(* CODESYS project Dual Magazijn Structured Text 2V0 - Demo 3V5SP13.project
   Company: Avans
   Description: Simulatie voor opstelling Sorteer Station.
   Title: Simulatie Sorteer Station
   Author: Rene Potters/Gerard Harkema
   Version: 0.1.0

Project tree, tasks and I/O mapping:
  Device_1 : CODESYS Control Win V3, 3S - Smart Software Solutions GmbH, version 3.5.13.20
    application MagazijnTestSimulatie
      libraries: Standard, * (System); Util, * (System); VisuDialogs, 3.5.16.40 (System)
      task MainTask (cyclic, interval t#20ms, priority 1) calls MagazijnTest
      task Simulatie (cyclic, interval t#20ms, priority 1) calls MagazijnSim1, MagazijnSim2
  Simulatie/
    program MagazijnSim1 [ST]
    global variables SIM1
    data type MagazijnDUT
    program MagazijnSim2 [ST]
    global variables SIM2
  text list GlobalTextList
  Programma Structured Text/
    function block MagazijnClass [ST]: initialize, cycle, start, isMagazijnLeeg, isError, reset, isKlaar, noodstop
    TestProgramms/
      program MagazijnTest [ST]
    States/
      data type magazijnStates
  global variables GVL1
  Visualisaties/
    visualisation BekerMagazijnHMI
  global variables GVL2
*)

// Simulatie/MagazijnDUT
{attribute 'qualified_only'}
{attribute 'strict'}
TYPE MagazijnDUT :
(
	INGETROKKEN, INTREKKEN, UITGESTOTEN, UITSTOTEN, LEEG
);
END_TYPE

// Programma Structured Text/States/magazijnStates
// Datum : 17 december 2020, Auteur: Gerard Harkema
{attribute 'qualified_only'}
{attribute 'strict'}
TYPE magazijnStates :
(
	idle := 0,
	in,
	travel_out,
	out,
	travel_in,
	error
);
END_TYPE

// Simulatie/SIM1
{attribute 'qualified_only'}
VAR_GLOBAL
	// Rotatie van de overzetter
	Vx_OvzRotate: INT := 0;
	// Visualisatie invisible blok
	Vx_OvzBlokLinks: BOOL := FALSE;
	// Visualisatie invisible blok
	Vx_OvzBlokOverzetter: BOOL := FALSE;
	// Visualisatie invisible blok
	Vx_OvzBlokRechts: BOOL := FALSE;
	// Visualisatie invisible blok
	Vx_OvzBlokGevallen: BOOL := FALSE;	
	// Magazijn opnieuw vullen (simulatie)
	Ix_MagazijnVullen 	: BOOL;
	// Goten legen (symulatie)
	Ix_GotenLegen	  	: BOOL;
	
	
	
	
	
	
	
	
	
	
	
	
	
	
	
	
	
	
	
	
	
	
	
	
	
	
	
	
	
	
	
	
	
	
	
	
	
	
	
	
	
	
	
	
	
	
	
	
	// Simulatie visualisatie 
	Vw_Rotate45: INT := 45;
	// Visualisatie X positie van de uitstoter
	Vw_MagUitstoterBekerX: INT := 30;
	// Visualisatie invisible blok uitgestoten
	Vx_MagBlokUit: BOOL := TRUE;
	// Visualisatie invisible blok 1
	Vx_MagBlok1: BOOL := TRUE;
	// Visualisatie invisible blok 2
	Vx_MagBlok2: BOOL := TRUE;
	// Visualisatie invisible blok 3
	Vx_MagBlok3: BOOL := TRUE;
	// Visualisatie invisible blok 4
	Vx_MagBlok4: BOOL := TRUE;
	// Visualisatie invisible blokken
	Vx_MagBlok: ARRAY[1..8] OF BOOL;
	// Aantal blokken in het magazijn
	Vw_MagBlokAantal: INT := 4;
	// Simulatie onthoudt dat een blok maar 1x wordt uitgestoten
	Vw_MagBlok1X: INT := 0;
	// Ligt er een blok op band
	Vw_SorBlokBand: BOOL := FALSE;
	// Rotatie van de stopper
	Vw_SorStopperRotate: INT := 0;
	// Rotatie van de stopper goot 1
	Vw_SorGoot1Rotate: INT := 0;
	// Rotatie van de stopper goot 2
	Vw_SorGoot2Rotate: INT := 0;
	// Kleur van de blok op betreffende positie
	Vw_SorKleurBand: DWORD := 0;
	// Bewegen van de blok over de band
	Vi_SorBlokBandX: INT := 0;
	// Bewegen van de blok over de band
	Vi_SorBlokBandY: INT := 0;
	// Simulatie error. Inverse logica.
	Vx_MagLuchtDrukError: BOOL := TRUE;
	// Simulatie error. Inverse logica.
	Vx_MagIsInError: BOOL := TRUE;
	// Simulatie error. Inverse logica.
	Vx_MagIsUitError: BOOL := TRUE;
	// Simulatie error. Inverse logica.
	Vx_OvzLuchtDrukError: BOOL := TRUE;
	// Simulatie error. Inverse logica.
	Vx_OvzIsLinksError: BOOL := TRUE;
	// Simulatie error. Inverse logica.
	Vx_OvzIsRechtsError: BOOL := TRUE;
	// Simulatie error. Inverse logica.
	Vx_OvzVacuumError: BOOL := TRUE;
	// Simulatie error. Inverse logica.
	Vx_SorMotorAfvoerError: BOOL := TRUE;
	// Simulatie error. Inverse logica.
	Vx_SorGoot1InError: BOOL := TRUE;
	// Simulatie error. Inverse logica.
	Vx_SorGoot1UitError: BOOL := TRUE;
	// Simulatie error. Inverse logica.
	Vx_SorInGootError: BOOL := TRUE;
	// Ligt er een blok op de betreffende positie
	Vx_SorBlokGoot: ARRAY [1..3,1..6] OF BOOL;
	// Kleur van de blok op betreffende positie
	Vw_SorKleurGoot: ARRAY [1..3,1..6] OF DWORD;
END_VAR

// GVL1
VAR_GLOBAL
	// Indrukken resetknop 
	Ix_Resetknop: BOOL;
	// Keuzeknop staat op hand
	Ix_Hand: BOOL;
	// Keuzeknop staat op auto
	Ix_Auto: BOOL;
	// Indrukken noodstop
	Ix_Noodstop: BOOL;
	// Bekers magazijn zijn op
	Ix_MagazijnLeeg: BOOL;
	// Beker is uit dekselmagazijn gestoten
	Ix_UitstoterBekerIn: BOOL;
	// Uitstoter Beker haalt nieuwe beker op
	Ix_UitstoterBekerUit: BOOL;
	// Indrukken startknop
	Ix_Stopknop: BOOL := TRUE;
	// Indrukken stopknop
	Ix_Startknop: BOOL;	
	//Perslucht is aanwezig
	Ix_PersluchtAanwezig :BOOL;
	//Werkstuk door overzetter opgepakt
	Ix_VacuumAanwezig :BOOL;
	//Overzetter haalt beker op(linker pos.)
	Ix_OverzetterIsLinks :BOOL;
	//Overzetter plaatst beker op sorteerpositie
	Ix_OverzetterIsRechts :BOOL;
	//Beker aanwezig op detectiepositie
	Ix_BekerAanwezig :BOOL;
	//Beker is van aluminium
	Ix_BekerMetaal :BOOL;
	//Beker reflecteert en is dus niet zwart
	Ix_BekerReflecteerd :BOOL;
	//Product is naar een van de goten gegaan
	Ix_BekerInGoot :BOOL;
	//Pusher uitvoergoot 1 is in
	Ix_UitvoerGoot1IsIn :BOOL;
	//Pusher uitvoergoot 2 is in
	Ix_UitvoerGoot2IsIn :BOOL;
	//Beker afvoeren is bezig
	Ix_StationAfvoerVrij :BOOL;
	//Pusher uitvoergoot 1 is uit
	Ix_UitvoerGoot1IsUit :BOOL;
	//Pusher uitvoergoot 2 is uit
	Ix_UitvoerGoot2IsUit :BOOL;
	// Beker uit magazijn stoten
	Qx_BekerUitstoten: BOOL;	
	//Beker oppakken
	Qx_VacuumAan :BOOL;
	//Beker loslaten
	Qx_BekerLossen :BOOL;
	//Overzetter naar bekermagazijn
	Qx_OverzetterLinks :BOOL;
	//Overzetter naar sorteerpositie
	Qx_OverzetterRechts :BOOL;
	//Transportband aan
	Qx_MotorAfvoerAan :BOOL;
	//Pusher goot 1 uit
	Qx_UitvoerGoot1Uit :BOOL;
	//Pusher goot 2 uit
	Qx_UitvoerGoot2Uit :BOOL;
	//Beker stoppen op band voor detectie
	Qx_StopperUit :BOOL;
	//Uitsorteren is bezet
	Qx_StationBezet :BOOL;
	// Visualisatie invisible Gele vlak
	Qx_GeleLamp: BOOL;
	// Visualisatie invisible groene vlak
	Qx_GroeneLamp: BOOL;
	// Visualisatie invisible rode vlak
	Qx_RodeLamp: BOOL;
END_VAR

// Simulatie/SIM2
{attribute 'qualified_only'}
VAR_GLOBAL
	// Rotatie van de overzetter
	Vx_OvzRotate: INT := 0;
	// Visualisatie invisible blok
	Vx_OvzBlokLinks: BOOL := FALSE;
	// Visualisatie invisible blok
	Vx_OvzBlokOverzetter: BOOL := FALSE;
	// Visualisatie invisible blok
	Vx_OvzBlokRechts: BOOL := FALSE;
	// Visualisatie invisible blok
	Vx_OvzBlokGevallen: BOOL := FALSE;	
	// Magazijn opnieuw vullen (simulatie)
	Ix_MagazijnVullen 	: BOOL;
	// Goten legen (symulatie)
	Ix_GotenLegen	  	: BOOL;
	
	
	
	
	
	
	
	
	
	
	
	
	
	
	
	
	
	
	
	
	
	
	
	
	
	
	
	
	
	
	
	
	
	
	
	
	
	
	
	
	
	
	
	
	
	
	
	
	// Simulatie visualisatie 
	Vw_Rotate45: INT := 45;
	// Visualisatie X positie van de uitstoter
	Vw_MagUitstoterBekerX: INT := 30;
	// Visualisatie invisible blok uitgestoten
	Vx_MagBlokUit: BOOL := TRUE;
	// Visualisatie invisible blok 1
	Vx_MagBlok1: BOOL := TRUE;
	// Visualisatie invisible blok 2
	Vx_MagBlok2: BOOL := TRUE;
	// Visualisatie invisible blok 3
	Vx_MagBlok3: BOOL := TRUE;
	// Visualisatie invisible blok 4
	Vx_MagBlok4: BOOL := TRUE;
	// Visualisatie invisible blokken
	Vx_MagBlok: ARRAY[1..8] OF BOOL;
	// Aantal blokken in het magazijn
	Vw_MagBlokAantal: INT := 4;
	// Simulatie onthoudt dat een blok maar 1x wordt uitgestoten
	Vw_MagBlok1X: INT := 0;
	// Ligt er een blok op band
	Vw_SorBlokBand: BOOL := FALSE;
	// Rotatie van de stopper
	Vw_SorStopperRotate: INT := 0;
	// Rotatie van de stopper goot 1
	Vw_SorGoot1Rotate: INT := 0;
	// Rotatie van de stopper goot 2
	Vw_SorGoot2Rotate: INT := 0;
	// Kleur van de blok op betreffende positie
	Vw_SorKleurBand: DWORD := 0;
	// Bewegen van de blok over de band
	Vi_SorBlokBandX: INT := 0;
	// Bewegen van de blok over de band
	Vi_SorBlokBandY: INT := 0;
	// Simulatie error. Inverse logica.
	Vx_MagLuchtDrukError: BOOL := TRUE;
	// Simulatie error. Inverse logica.
	Vx_MagIsInError: BOOL := TRUE;
	// Simulatie error. Inverse logica.
	Vx_MagIsUitError: BOOL := TRUE;
	// Simulatie error. Inverse logica.
	Vx_OvzLuchtDrukError: BOOL := TRUE;
	// Simulatie error. Inverse logica.
	Vx_OvzIsLinksError: BOOL := TRUE;
	// Simulatie error. Inverse logica.
	Vx_OvzIsRechtsError: BOOL := TRUE;
	// Simulatie error. Inverse logica.
	Vx_OvzVacuumError: BOOL := TRUE;
	// Simulatie error. Inverse logica.
	Vx_SorMotorAfvoerError: BOOL := TRUE;
	// Simulatie error. Inverse logica.
	Vx_SorGoot1InError: BOOL := TRUE;
	// Simulatie error. Inverse logica.
	Vx_SorGoot1UitError: BOOL := TRUE;
	// Simulatie error. Inverse logica.
	Vx_SorInGootError: BOOL := TRUE;
	// Ligt er een blok op de betreffende positie
	Vx_SorBlokGoot: ARRAY [1..3,1..6] OF BOOL;
	// Kleur van de blok op betreffende positie
	Vw_SorKleurGoot: ARRAY [1..3,1..6] OF DWORD;
END_VAR

// GVL2
VAR_GLOBAL
	// Indrukken resetknop 
	Ix_Resetknop: BOOL;
	// Keuzeknop staat op hand
	Ix_Hand: BOOL;
	// Keuzeknop staat op auto
	Ix_Auto: BOOL;
	// Indrukken noodstop
	Ix_Noodstop: BOOL;
	// Bekers magazijn zijn op
	Ix_MagazijnLeeg: BOOL;
	// Beker is uit dekselmagazijn gestoten
	Ix_UitstoterBekerIn: BOOL;
	// Uitstoter Beker haalt nieuwe beker op
	Ix_UitstoterBekerUit: BOOL;
	// Indrukken startknop
	Ix_Stopknop: BOOL := TRUE;
	// Indrukken stopknop
	Ix_Startknop: BOOL;	
	//Perslucht is aanwezig
	Ix_PersluchtAanwezig :BOOL;
	//Werkstuk door overzetter opgepakt
	Ix_VacuumAanwezig :BOOL;
	//Overzetter haalt beker op(linker pos.)
	Ix_OverzetterIsLinks :BOOL;
	//Overzetter plaatst beker op sorteerpositie
	Ix_OverzetterIsRechts :BOOL;
	//Beker aanwezig op detectiepositie
	Ix_BekerAanwezig :BOOL;
	//Beker is van aluminium
	Ix_BekerMetaal :BOOL;
	//Beker reflecteert en is dus niet zwart
	Ix_BekerReflecteerd :BOOL;
	//Product is naar een van de goten gegaan
	Ix_BekerInGoot :BOOL;
	//Pusher uitvoergoot 1 is in
	Ix_UitvoerGoot1IsIn :BOOL;
	//Pusher uitvoergoot 2 is in
	Ix_UitvoerGoot2IsIn :BOOL;
	//Beker afvoeren is bezig
	Ix_StationAfvoerVrij :BOOL;
	//Pusher uitvoergoot 1 is uit
	Ix_UitvoerGoot1IsUit :BOOL;
	//Pusher uitvoergoot 2 is uit
	Ix_UitvoerGoot2IsUit :BOOL;
	// Beker uit magazijn stoten
	Qx_BekerUitstoten: BOOL;	
	//Beker oppakken
	Qx_VacuumAan :BOOL;
	//Beker loslaten
	Qx_BekerLossen :BOOL;
	//Overzetter naar bekermagazijn
	Qx_OverzetterLinks :BOOL;
	//Overzetter naar sorteerpositie
	Qx_OverzetterRechts :BOOL;
	//Transportband aan
	Qx_MotorAfvoerAan :BOOL;
	//Pusher goot 1 uit
	Qx_UitvoerGoot1Uit :BOOL;
	//Pusher goot 2 uit
	Qx_UitvoerGoot2Uit :BOOL;
	//Beker stoppen op band voor detectie
	Qx_StopperUit :BOOL;
	//Uitsorteren is bezet
	Qx_StationBezet :BOOL;
	// Visualisatie invisible Gele vlak
	Qx_GeleLamp: BOOL;
	// Visualisatie invisible groene vlak
	Qx_GroeneLamp: BOOL;
	// Visualisatie invisible rode vlak
	Qx_RodeLamp: BOOL;
END_VAR

// Programma Structured Text/TestProgramms/MagazijnTest
// Datum : 17 december 2020, Auteur: Gerard Harkema
PROGRAM MagazijnTest
VAR
	xInitialaized				: BOOL := FALSE;
	
	// Bekers magazijn zijn op
	Ix_MagazijnLeegRef1			: REFERENCE TO BOOL;
	// Beker is uit dekselmagazijn gestoten
	Ix_UitstoterBekerInRef1		: REFERENCE TO BOOL;
	// Uitstoter Beker haalt nieuwe beker op
	Ix_UitstoterBekerUitRef1	: REFERENCE TO BOOL;
	// Beker uit magazijn stoten
	Qx_BekerUitstotenRef1		: REFERENCE TO BOOL;
	
	// Bekers magazijn zijn op
	Ix_MagazijnLeegRef2			: REFERENCE TO BOOL;
	// Beker is uit dekselmagazijn gestoten
	Ix_UitstoterBekerInRef2		: REFERENCE TO BOOL;
	// Uitstoter Beker haalt nieuwe beker op
	Ix_UitstoterBekerUitRef2	: REFERENCE TO BOOL;
	// Beker uit magazijn stoten
	Qx_BekerUitstotenRef2		: REFERENCE TO BOOL;

	magazijn1: MagazijnClass;
	magazijn2: MagazijnClass;
	
END_VAR

IF NOT xInitialaized THEN

	// Forse Persluct aanwezig
	GVL1.Ix_PersluchtAanwezig := TRUE;
	
	Ix_MagazijnLeegRef1 		REF= GVL1.Ix_MagazijnLeeg;
	Ix_UitstoterBekerInRef1 	REF= GVL1.Ix_UitstoterBekerIn;
	Ix_UitstoterBekerUitRef1 	REF= GVL1.Ix_UitstoterBekerUit;
	Qx_BekerUitstotenRef1 		REF= GVL1.Qx_BekerUitstoten;

	magazijn1.initialize(Ix_MagazijnLeegRef1,
					    Ix_UitstoterBekerInRef1,
						Ix_UitstoterBekerUitRef1,
						Qx_BekerUitstotenRef1,
						GVL1.Ix_PersluchtAanwezig);
	
	Ix_MagazijnLeegRef2 		REF= GVL2.Ix_MagazijnLeeg;
	Ix_UitstoterBekerInRef2 	REF= GVL2.Ix_UitstoterBekerIn;
	Ix_UitstoterBekerUitRef2 	REF= GVL2.Ix_UitstoterBekerUit;
	Qx_BekerUitstotenRef2 		REF= GVL2.Qx_BekerUitstoten;

	magazijn2.initialize(Ix_MagazijnLeegRef2,
					    Ix_UitstoterBekerInRef2,
						Ix_UitstoterBekerUitRef2,
						Qx_BekerUitstotenRef2,
						GVL1.Ix_PersluchtAanwezig);
						
						
	xInitialaized	:= TRUE;
END_IF

IF GVL1.Ix_Startknop THEN
	magazijn1.start();
	GVL1.Ix_Startknop := FALSE;
END_IF

IF GVL1.Ix_Resetknop THEN
	magazijn1.reset();
END_IF

IF GVL1.Ix_Noodstop THEN
	magazijn1.noodstop();
END_IF

GVL1.Qx_GroeneLamp := magazijn1.isKlaar();
GVL1.Qx_RodeLamp := magazijn1.isError();
GVL1.Qx_GeleLamp := magazijn1.isMagazijnLeeg();
 
IF GVL2.Ix_Startknop THEN
	magazijn2.start();
	GVL2.Ix_Startknop := FALSE;
END_IF

IF GVL2.Ix_Resetknop THEN
	magazijn2.reset();
END_IF

IF GVL2.Ix_Noodstop THEN
	magazijn2.noodstop();
END_IF

GVL2.Qx_GroeneLamp := magazijn2.isKlaar();
GVL2.Qx_RodeLamp := magazijn2.isError();
GVL2.Qx_GeleLamp := magazijn2.isMagazijnLeeg();

magazijn1.cycle();
magazijn2.cycle();

END_PROGRAM

// Programma Structured Text/MagazijnClass
// Datum : 17 december 2020, Auteur: Gerard Harkema
FUNCTION_BLOCK MagazijnClass
VAR
	// Bekers magazijn zijn op
	Ix_MagazijnLeeg				: REFERENCE TO BOOL;
	// Beker is uit dekselmagazijn gestoten
	Ix_UitstoterBekerIn			: REFERENCE TO BOOL;
	// Uitstoter Beker haalt nieuwe beker op
	Ix_UitstoterBekerUit		: REFERENCE TO BOOL;
	// Beker uit magazijn stoten
	Qx_BekerUitstoten			: REFERENCE TO BOOL;

	//Perslucht is aanwezig
	Ix_PersluchtAanwezig 		: REFERENCE TO BOOL;

	xInitialized				: BOOL := FALSE;
	xKlaar						: BOOL := FALSE;
	eState 						: magazijnStates := magazijnStates.idle;
	
END_VAR

IF NOT xInitialized THEN

	xInitialized				:= TRUE;

END_IF

// Datum : 17 december 2020, Auteur: Gerard Harkema
METHOD initialize
VAR_INPUT
	// Bekers magazijn zijn op
	Ix_MagazijnLeegRef		: REFERENCE TO BOOL;
	// Beker is uit dekselmagazijn gestoten
	Ix_UitstoterBekerInRef	: REFERENCE TO BOOL;
	// Uitstoter Beker haalt nieuwe beker op
	Ix_UitstoterBekerUitRef	: REFERENCE TO BOOL;
	// Beker uit magazijn stoten
	Qx_BekerUitstotenRef	: REFERENCE TO BOOL;
	
	//Perslucht is aanwezig
	Ix_PersluchtAanwezigRef : REFERENCE TO BOOL;

END_VAR
// Bekers magazijn zijn op
Ix_MagazijnLeeg 			REF= Ix_MagazijnLeegRef;
// Beker is uit dekselmagazijn gestoten
Ix_UitstoterBekerIn 		REF= Ix_UitstoterBekerInRef;
// Uitstoter Beker haalt nieuwe beker op
Ix_UitstoterBekerUit 		REF= Ix_UitstoterBekerUitRef;
// Beker uit magazijn stoten
Qx_BekerUitstoten 			REF= Qx_BekerUitstotenRef;
//Perslucht is aanwezig
Ix_PersluchtAanwezig 		REF= Ix_PersluchtAanwezigRef;

eState 						:= magazijnStates.travel_in;
END_METHOD

// Datum : 17 december 2020, Auteur: Gerard Harkema
METHOD cycle
VAR_INPUT
END_VAR

CASE eState OF
	//magazijnStates.idle:
	//magazijnStates.in:
	magazijnStates.travel_out:
		IF Ix_UitstoterBekerUit THEN
			eState 			:= magazijnStates.out;	
			Qx_BekerUitstoten 	:= FALSE;
		END_IF
	magazijnStates.out:
		eState 				:= magazijnStates.travel_in;	
	magazijnStates.travel_in:
		IF Ix_UitstoterBekerIn THEN
			eState 			:= magazijnStates.in;
			xKlaar			:= True;	
		END_IF
	
	//magazijnStates.error:
END_CASE
END_METHOD

// Datum : 17 december 2020, Auteur: Gerard Harkema
METHOD start : BOOL
VAR_INPUT
END_VAR
IF isMagazijnLeeg() THEN
	eState 				:= magazijnStates.error;
	Qx_BekerUitstoten 	:= FALSE;
	start 		:= TRUE; // Failed
	RETURN;
END_IF

IF NOT Ix_PersluchtAanwezig THEN
	eState 				:= magazijnStates.error;
	Qx_BekerUitstoten 	:= FALSE;
	start 		:= TRUE; // Failed
	RETURN;
END_IF

IF NOT (eState = magazijnStates.in) THEN
	eState 				:= magazijnStates.error;
	Qx_BekerUitstoten 	:= FALSE;
	start 		:= TRUE; // Failed
	RETURN;	
END_IF

xKlaar 					:= FALSE;
Qx_BekerUitstoten 		:= TRUE;
eState 					:= magazijnStates.travel_out;

start 			:= FALSE; // oké
END_METHOD

// Datum : 17 december 2020, Auteur: Gerard Harkema
METHOD isMagazijnLeeg : BOOL
VAR_INPUT
END_VAR
isMagazijnLeeg := Ix_MagazijnLeeg;
END_METHOD

// Datum : 17 december 2020, Auteur: Gerard Harkema
METHOD isError : BOOL
VAR_INPUT
END_VAR
isError := (eState = magazijnStates.error);
END_METHOD

// Datum : 17 december 2020, Auteur: Gerard Harkema
METHOD reset : BOOL
VAR_INPUT
END_VAR
eState 		:= magazijnStates.travel_in;
END_METHOD

// Datum : 17 december 2020, Auteur: Gerard Harkema
METHOD isKlaar : BOOL
VAR_INPUT
END_VAR
isKlaar := xKlaar;
END_METHOD

// Datum : 17 december 2020, Auteur: Gerard Harkema
METHOD noodstop
VAR_INPUT
END_VAR
eState 				:= magazijnStates.error;
Qx_BekerUitstoten 	:= FALSE;
END_METHOD

END_FUNCTION_BLOCK

// Simulatie/MagazijnSim1
PROGRAM MagazijnSim1
VAR
	// Timer om uitstoten en intrekken te vertragen
	Fb_Pulse: BLINK;
	// Timer om intrekken te vertragen
	Fb_Trigger: F_TRIG;
	// Eerste keer om visualisatie te updaten
	Mx_FirstTime: BOOL := TRUE;
	// Afhandeling van het magazijn
	Me_MagState: MAGAZIJNDUT := MAGAZIJNDUT.INGETROKKEN;
END_VAR

//
// Common stuff.
//

IF (Mx_FirstTime) THEN
	SIM1.Vw_MagBlokAantal := 8;
	SIM1.Vx_MagBlokUit:= FALSE;
	
	Mx_FirstTime := FALSE;
END_IF

					
//
// Handle all pulse and trigger events.
//
Fb_Pulse(ENABLE:=TRUE,TIMELOW:=T#200MS, TIMEHIGH:=T#200MS);
Fb_Trigger(CLK:=Fb_Pulse.OUT);


//
// Only if no emergency active, start handling the simulation.
//
IF (SIM1.Ix_MagazijnVullen) THEN
	Mx_FirstTime := TRUE;
	SIM1.Ix_MagazijnVullen := FALSE;
	RETURN;
END_IF
	
//
// The pulse determines the speed of the cilinder to move in
// ore move out. The cilinder is only moved if the airpressure 
// is available.
//
IF (Fb_Trigger.Q AND SIM1.Vx_MagLuchtDrukError) THEN
		
			
	CASE Me_MagState OF
		MAGAZIJNDUT.INGETROKKEN:
			IF (SIM1.Vx_MagBlokUit) THEN
				SIM1.Vw_MagBlokAantal := SIM1.Vw_MagBlokAantal - 1;
			END_IF
		
			SIM1.Vw_MagUitstoterBekerX := 1;
			SIM1.Vw_MagBlok1X    	  := SIM1.Vw_MagUitstoterBekerX;
			SIM1.Vx_MagBlokUit         := FALSE;
	
			IF (GVL1.Qx_BekerUitstoten) THEN
				Me_MagState := MAGAZIJNDUT.UITSTOTEN;
			END_IF

		MAGAZIJNDUT.INTREKKEN:
			SIM1.Vw_MagUitstoterBekerX := SIM1.Vw_MagUitstoterBekerX - 30;
			
			IF (SIM1.Vw_MagUitstoterBekerX < 0) THEN 
				SIM1.Vw_MagUitstoterBekerX := 0; 
			END_IF		
			
			IF (SIM1.Vw_MagUitstoterBekerX = 0) THEN
				Me_MagState := MAGAZIJNDUT.INGETROKKEN;				
			END_IF		

			IF (GVL1.Qx_BekerUitstoten) THEN
				Me_MagState := MAGAZIJNDUT.UITSTOTEN;
			END_IF	
	
		MAGAZIJNDUT.UITGESTOTEN:
			SIM1.Vx_MagBlokUit         := SIM1.Vx_MagBlok1;
						
			IF (NOT GVL1.Qx_BekerUitstoten) THEN
				Me_MagState := MAGAZIJNDUT.INTREKKEN;
			END_IF	
		
		MAGAZIJNDUT.UITSTOTEN:
			SIM1.Vw_MagUitstoterBekerX := SIM1.Vw_MagUitstoterBekerX + 30;
			SIM1.Vw_MagBlok1X    	  := SIM1.Vw_MagUitstoterBekerX;			
		
			IF (SIM1.Vw_MagUitstoterBekerX > 70) THEN
				Me_MagState := MAGAZIJNDUT.UITGESTOTEN;				
			END_IF		

			IF (NOT GVL1.Qx_BekerUitstoten) THEN
				Me_MagState := MAGAZIJNDUT.INTREKKEN;
			END_IF	
		
	END_CASE

	GVL1.Ix_UitstoterBekerIn  := (Me_MagState = MAGAZIJNDUT.INGETROKKEN) AND SIM1.Vx_MagIsInError;
	GVL1.Ix_UitstoterBekerUit := (Me_MagState = MAGAZIJNDUT.UITGESTOTEN) AND SIM1.Vx_MagIsUitError;	
	GVL1.Ix_MagazijnLeeg 	 := (SIM1.Vw_MagBlokAantal <= 0) AND (GVL1.Ix_UitstoterBekerIn);	
	
	SIM1.Vx_MagBlok[8] := (SIM1.Vw_MagBlokAantal >= 8);
	SIM1.Vx_MagBlok[7] := (SIM1.Vw_MagBlokAantal >= 7);
	SIM1.Vx_MagBlok[6] := (SIM1.Vw_MagBlokAantal >= 6);
	SIM1.Vx_MagBlok[5] := (SIM1.Vw_MagBlokAantal >= 5);		
	SIM1.Vx_MagBlok[4] := (SIM1.Vw_MagBlokAantal >= 4);
	SIM1.Vx_MagBlok[3] := (SIM1.Vw_MagBlokAantal >= 3);
	SIM1.Vx_MagBlok[2] := (SIM1.Vw_MagBlokAantal >= 2);
	SIM1.Vx_MagBlok[1] := (SIM1.Vw_MagBlokAantal >= 1);	
	
END_IF

END_PROGRAM

// Simulatie/MagazijnSim2
PROGRAM MagazijnSim2
VAR
	// Timer om uitstoten en intrekken te vertragen
	Fb_Pulse: BLINK;
	// Timer om intrekken te vertragen
	Fb_Trigger: F_TRIG;
	// Eerste keer om visualisatie te updaten
	Mx_FirstTime: BOOL := TRUE;
	// Afhandeling van het magazijn
	Me_MagState: MAGAZIJNDUT := MAGAZIJNDUT.INGETROKKEN;
END_VAR

//
// Common stuff.
//

IF (Mx_FirstTime) THEN
	SIM2.Vw_MagBlokAantal := 8;
	SIM2.Vx_MagBlokUit:= FALSE;
	
	Mx_FirstTime := FALSE;
END_IF

					
//
// Handle all pulse and trigger events.
//
Fb_Pulse(ENABLE:=TRUE,TIMELOW:=T#200MS, TIMEHIGH:=T#200MS);
Fb_Trigger(CLK:=Fb_Pulse.OUT);


//
// Only if no emergency active, start handling the simulation.
//
IF (SIM2.Ix_MagazijnVullen) THEN
	Mx_FirstTime := TRUE;
	SIM2.Ix_MagazijnVullen := FALSE;
	RETURN;
END_IF
	
//
// The pulse determines the speed of the cilinder to move in
// ore move out. The cilinder is only moved if the airpressure 
// is available.
//
IF (Fb_Trigger.Q AND SIM2.Vx_MagLuchtDrukError) THEN
		
			
	CASE Me_MagState OF
		MAGAZIJNDUT.INGETROKKEN:
			IF (SIM2.Vx_MagBlokUit) THEN
				SIM2.Vw_MagBlokAantal := SIM2.Vw_MagBlokAantal - 1;
			END_IF
		
			SIM2.Vw_MagUitstoterBekerX := 1;
			SIM2.Vw_MagBlok1X    	  := SIM2.Vw_MagUitstoterBekerX;
			SIM2.Vx_MagBlokUit         := FALSE;
	
			IF (GVL2.Qx_BekerUitstoten) THEN
				Me_MagState := MAGAZIJNDUT.UITSTOTEN;
			END_IF

		MAGAZIJNDUT.INTREKKEN:
			SIM2.Vw_MagUitstoterBekerX := SIM2.Vw_MagUitstoterBekerX - 30;
			
			IF (SIM2.Vw_MagUitstoterBekerX < 0) THEN 
				SIM2.Vw_MagUitstoterBekerX := 0; 
			END_IF		
			
			IF (SIM2.Vw_MagUitstoterBekerX = 0) THEN
				Me_MagState := MAGAZIJNDUT.INGETROKKEN;				
			END_IF		

			IF (GVL2.Qx_BekerUitstoten) THEN
				Me_MagState := MAGAZIJNDUT.UITSTOTEN;
			END_IF	
	
		MAGAZIJNDUT.UITGESTOTEN:
			SIM2.Vx_MagBlokUit         := SIM2.Vx_MagBlok1;
						
			IF (NOT GVL2.Qx_BekerUitstoten) THEN
				Me_MagState := MAGAZIJNDUT.INTREKKEN;
			END_IF	
		
		MAGAZIJNDUT.UITSTOTEN:
			SIM2.Vw_MagUitstoterBekerX := SIM2.Vw_MagUitstoterBekerX + 30;
			SIM2.Vw_MagBlok1X    	  := SIM2.Vw_MagUitstoterBekerX;			
		
			IF (SIM2.Vw_MagUitstoterBekerX > 70) THEN
				Me_MagState := MAGAZIJNDUT.UITGESTOTEN;				
			END_IF		

			IF (NOT GVL2.Qx_BekerUitstoten) THEN
				Me_MagState := MAGAZIJNDUT.INTREKKEN;
			END_IF	
		
	END_CASE

	GVL2.Ix_UitstoterBekerIn  := (Me_MagState = MAGAZIJNDUT.INGETROKKEN) AND SIM2.Vx_MagIsInError;
	GVL2.Ix_UitstoterBekerUit := (Me_MagState = MAGAZIJNDUT.UITGESTOTEN) AND SIM2.Vx_MagIsUitError;	
	GVL2.Ix_MagazijnLeeg 	 := (SIM2.Vw_MagBlokAantal <= 0) AND (GVL2.Ix_UitstoterBekerIn);	
	
	SIM2.Vx_MagBlok[8] := (SIM2.Vw_MagBlokAantal >= 8);
	SIM2.Vx_MagBlok[7] := (SIM2.Vw_MagBlokAantal >= 7);
	SIM2.Vx_MagBlok[6] := (SIM2.Vw_MagBlokAantal >= 6);
	SIM2.Vx_MagBlok[5] := (SIM2.Vw_MagBlokAantal >= 5);		
	SIM2.Vx_MagBlok[4] := (SIM2.Vw_MagBlokAantal >= 4);
	SIM2.Vx_MagBlok[3] := (SIM2.Vw_MagBlokAantal >= 3);
	SIM2.Vx_MagBlok[2] := (SIM2.Vw_MagBlokAantal >= 2);
	SIM2.Vx_MagBlok[1] := (SIM2.Vw_MagBlokAantal >= 1);	
	
END_IF

END_PROGRAM

// Visualisaties/BekerMagazijnHMI
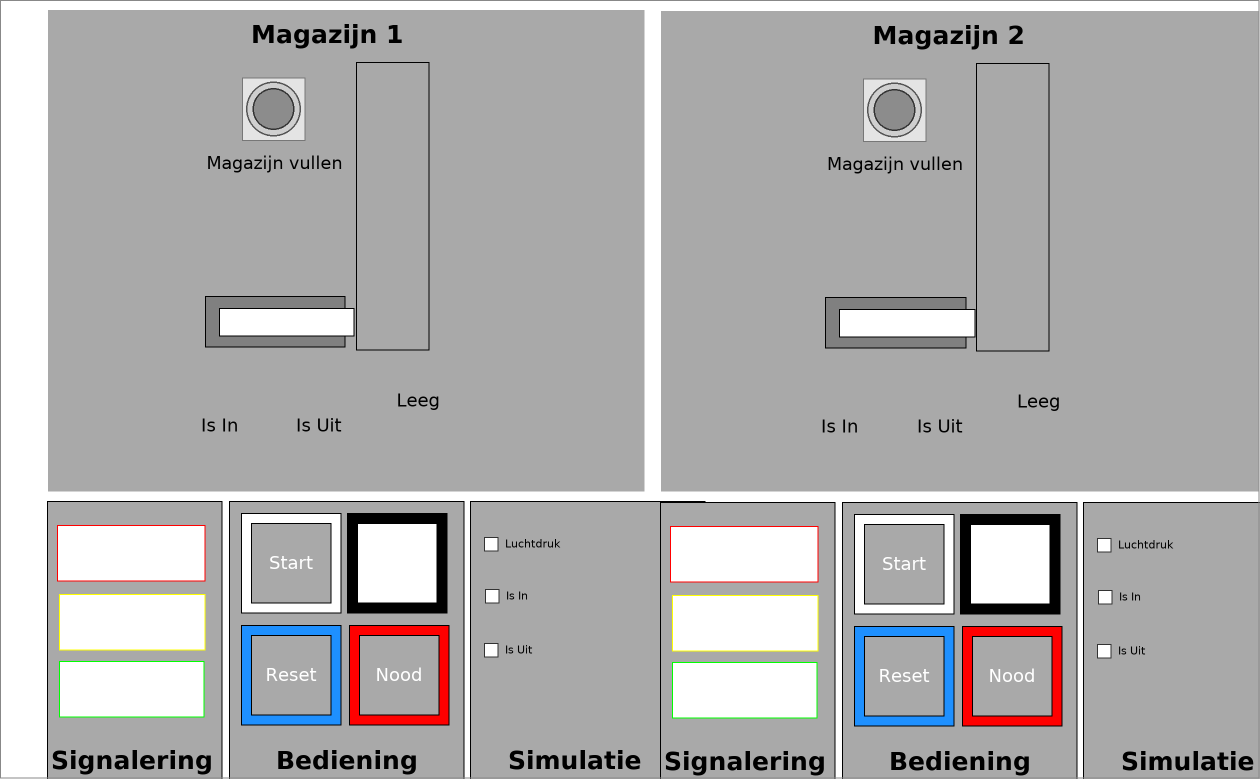
VISUALIZATION BekerMagazijnHMI  // 1260x779
    Group (47,9 1213x770)
        Group (0,0 599x769)
            Group (0,492 599x277)
                Group (0,0 173x277)
                    Rectangle (0,0 175x295)
                    Rectangle (10,24 148x56), colour toggle: GVL1.Qx_RodeLamp
                    Rectangle (12,93 146x56), colour toggle: GVL1.Qx_GeleLamp
                    Rectangle (12,160 145x56), colour toggle: GVL1.Qx_GroeneLamp
                    Label (10,236 150x46), "Signalering"
                Group (182,0 232x277)
                    Rectangle (0,0 235x295)
                    Group (12,12 100x100)
                        RoundedRectangle (0,0 100x100)
                        RoundedRectangle (10,10 80x80), "Start", tooltip "Start knop", colour toggle: GVL1.Ix_Startknop
                            OnMouseDown: execute { gvl1.Ix_Startknop := TRUE; }
                            OnMouseUp: execute { GVL1.Ix_Startknop := FALSE; }
                    Group (118,12 100x100)
                        RoundedRectangle (0,0 100x100)
                        RoundedRectangle (10,10 80x80), "Stop", tooltip "Stop knop", colour toggle: GVL1.Ix_Stopknop
                            OnMouseDown: execute { GVL1.Ix_Stopknop := FALSE; }
                            OnMouseUp: execute { GVL1.Ix_Stopknop := TRUE; }
                    Group (12,124 100x100)
                        RoundedRectangle (0,0 100x100)
                        RoundedRectangle (10,10 80x80), "Reset", tooltip "Reset knop", colour toggle: GVL1.Ix_Resetknop
                            OnMouseUp: execute { GVL1.Ix_Resetknop := FALSE; }
                    Group (120,124 100x100)
                        RoundedRectangle (0,0 100x100), "Nood"
                        RoundedRectangle (10,10 80x80), "Nood", tooltip "Noodstop", colour toggle: GVL1.Ix_Noodstop
                            OnMouseDown: execute { GVL1.Ix_Noodstop := NOT GVL1.Ix_Noodstop; }
                    Label (43,236 150x46), "Bediening"
                Group (423,0 176x277)
                    Group (0,0 235x295)
                        Rectangle (0,0 235x295)
                        Label (30,236 150x46), "Simulatie"
                    Checkbox (12,17 196x52), "Luchtdruk", variable: SIM1.Vx_MagLuchtDrukError
                    Checkbox (13,69 196x52), "Is In", variable: SIM1.Vx_MagIsInError
                    Checkbox (12,123 196x52), "Is Uit", variable: SIM1.Vx_MagIsUitError
            Group (0,0 598x483)
                Rectangle (0,0 598x483)
                Polygon (331,379) (358,379) (385,379) (412,379) (371,454), "Leeg", colour toggle: GVL1.Ix_MagazijnLeeg
                Polygon (173,379) (173,379) (209,417) (173,454) (137,417), "Is In", colour toggle: GVL1.Ix_UitstoterBekerIn
                Polygon (272,379) (272,379) (308,417) (272,454) (236,417), "Is Uit", colour toggle: GVL1.Ix_UitstoterBekerUit
                Rectangle (158,287 140x51)
                Rectangle (309,53 73x288)
                Rectangle (392,300 55x27), colour toggle: SIM1.Vx_MagBlokUit
                Rectangle (313,267 55x27), colour toggle: SIM1.Vx_MagBlok[2]
                Rectangle (313,233 55x27), colour toggle: SIM1.Vx_MagBlok[3]
                Rectangle (313,199 55x27), colour toggle: SIM1.Vx_MagBlok[4]
                Rectangle (313,300 55x27), colour toggle: SIM1.Vx_MagBlok[1]
                    p3560616238: SIM1.Vw_MagBlok1X
                Rectangle (172,299 135x28)
                    p3560616238: SIM1.Vw_MagUitstoterBekerX
                Label (213,11 135x28), "Magazijn 1"
                Rectangle (313,132 55x27), colour toggle: SIM1.Vx_MagBlok[6]
                Rectangle (313,98 55x27), colour toggle: SIM1.Vx_MagBlok[7]
                Rectangle (313,64 55x27), colour toggle: SIM1.Vx_MagBlok[8]
                Rectangle (313,165 55x27), colour toggle: SIM1.Vx_MagBlok[5]
                PushSwitch (195,67 63x66), tooltip "Magazijn vullen", variable: SIM1.Ix_MagazijnVullen, behaviour: TOGGLE, style: Switch-PushSwitch-Gray
                Polygon (158,142) (185,142) (212,142) (297,156) (207,169), "Magazijn vullen", colour toggle: Ix_MagazijnLeeg
        Group (613,1 600x769)
            Group (0,492 600x277)
                Group (0,0 173x277)
                    Rectangle (0,0 175x295)
                    Rectangle (10,24 148x56), colour toggle: GVL2.Qx_RodeLamp
                    Rectangle (12,93 146x56), colour toggle: GVL2.Qx_GeleLamp
                    Rectangle (12,160 145x56), colour toggle: GVL2.Qx_GroeneLamp
                    Label (10,236 150x46), "Signalering"
                Group (182,0 232x277)
                    Rectangle (0,0 235x295)
                    Group (12,12 100x100)
                        RoundedRectangle (0,0 100x100)
                        RoundedRectangle (10,10 80x80), "Start", tooltip "Start knop", colour toggle: GVL2.Ix_Startknop
                            OnMouseDown: execute { GVL2.Ix_Startknop := TRUE; }
                            OnMouseUp: execute { GVL2.Ix_Startknop := FALSE; }
                    Group (118,12 100x100)
                        RoundedRectangle (0,0 100x100)
                        RoundedRectangle (10,10 80x80), "Stop", tooltip "Stop knop", colour toggle: GVL2.Ix_Stopknop
                            OnMouseDown: execute { GVL2.Ix_Stopknop := FALSE; }
                            OnMouseUp: execute { GVL2.Ix_Stopknop := TRUE; }
                    Group (12,124 100x100)
                        RoundedRectangle (0,0 100x100)
                        RoundedRectangle (10,10 80x80), "Reset", tooltip "Reset knop", colour toggle: GVL2.Ix_Resetknop
                            OnMouseDown: execute { GVL2.Ix_Resetknop := TRUE; }
                            OnMouseUp: execute { GVL2.Ix_Resetknop := FALSE; }
                    Group (120,124 100x100)
                        RoundedRectangle (0,0 100x100), "Nood"
                        RoundedRectangle (10,10 80x80), "Nood", tooltip "Noodstop", colour toggle: GVL2.Ix_Noodstop
                            OnMouseDown: execute { Ix_Noodstop := NOT Ix_Noodstop; }
                    Label (43,236 150x46), "Bediening"
                Group (423,0 177x277)
                    Rectangle (0,0 235x295)
                    Label (30,236 150x46), "Simulatie"
                    Checkbox (12,17 196x52), "Luchtdruk", variable: SIM2.Vx_MagLuchtDrukError
                    Checkbox (13,69 196x52), "Is In", variable: SIM2.Vx_MagIsInError
                    Checkbox (12,123 196x52), "Is Uit", variable: SIM2.Vx_MagIsUitError
            Group (0,0 600x482)
                Rectangle (0,0 600x482)
                Polygon (338,379) (366,379) (393,379) (420,379) (379,454), "Leeg", colour toggle: GVL2.Ix_MagazijnLeeg
                Polygon (180,379) (180,379) (216,417) (180,454) (144,417), "Is In", colour toggle: GVL2.Ix_UitstoterBekerIn
                Polygon (280,379) (280,379) (316,417) (280,454) (244,417), "Is Uit", colour toggle: GVL2.Ix_UitstoterBekerUit
                Rectangle (165,287 141x51)
                Rectangle (316,53 73x288)
                Rectangle (400,300 55x27), colour toggle: SIM2.Vx_MagBlokUit
                Rectangle (321,267 55x27), colour toggle: SIM2.Vx_MagBlok[2]
                Rectangle (321,233 55x27), colour toggle: SIM2.Vx_MagBlok[3]
                Rectangle (321,199 55x27), colour toggle: SIM2.Vx_MagBlok[4]
                Rectangle (321,300 55x27), colour toggle: SIM2.Vx_MagBlok[1]
                    p3560616238: SIM2.Vw_MagBlok1X
                Rectangle (179,299 136x28)
                    p3560616238: SIM2.Vw_MagUitstoterBekerX
                Label (214,11 150x28), "Magazijn 2"
                Rectangle (321,132 55x27), colour toggle: SIM2.Vx_MagBlok[6]
                Rectangle (321,98 55x27), colour toggle: SIM2.Vx_MagBlok[7]
                Rectangle (321,64 55x27), colour toggle: SIM2.Vx_MagBlok[8]
                Rectangle (321,165 55x27), colour toggle: SIM2.Vx_MagBlok[5]
                PushSwitch (203,67 63x66), tooltip "Magazijn vullen", variable: SIM2.Ix_MagazijnVullen, behaviour: TOGGLE, style: Switch-PushSwitch-Gray
                Polygon (165,142) (192,142) (219,142) (305,156) (215,169), "Magazijn vullen", colour toggle: Ix_MagazijnLeeg
END_VISUALIZATION
